INTERFACE I_ContainModules

METHOD DeregisterCyclic : RegistrationResult
VAR_INPUT
	Cyclic : I_Cyclic;
END_VAR
END_METHOD

METHOD DeregisterInitialize : RegistrationResult
VAR_INPUT
	Initializable : I_Initializable;
END_VAR
END_METHOD

METHOD DeregisterModule : RegistrationResult
VAR_INPUT
	Module : I_Module;
END_VAR
END_METHOD

PROPERTY Modules : I_ModuleCollection
GET
END_GET
END_PROPERTY

METHOD RegisterCyclic  : RegistrationResult
VAR_INPUT
	Cyclic : I_Cyclic;
END_VAR
END_METHOD

METHOD RegisterInitialize  : RegistrationResult
VAR_INPUT
	Initializable : I_Initializable;
END_VAR
END_METHOD

METHOD RegisterModule  : RegistrationResult
VAR_INPUT
	Module : I_Module;
END_VAR
END_METHOD

END_INTERFACE

(* stored: Version 1.1.0.1, ProductVersion 3.1.4026.18
   Itf I_ContainModules: Id {c14c7da0-b6c9-4ae1-b029-af7adfe80c60}
   Method DeregisterCyclic: Id {dc661aae-00ab-44cc-852c-bc30e0d16315}
   Method DeregisterInitialize: Id {0f2dbb57-83a4-46ec-8357-7d426099c550}
   Method DeregisterModule: Id {08e0ee68-a6e4-4b09-8b7e-29d755ea3584}
   Property Modules: Id {ae884636-2441-4698-8484-af07377b9085}
   Get Get: Id {5f40a626-59fb-4998-9608-4f2df4af4b70}
   Method RegisterCyclic: Id {ac88bc75-086a-46cd-8466-5ef365758e65}
   Method RegisterInitialize: Id {490bed12-8da5-4fed-a7bc-b1907cf06592}
   Method RegisterModule: Id {2782642e-e5eb-495c-91f3-7fbac14f41b9} *)
